(* IEC 61131-3 sources: crb-codesys/retrieval/output/codesys_repo/Proxy_Application/FUN, 9 files *)

(* ---- Proxy.st ---- *)
{attribute 'enable_dynamic_creation'}
FUNCTION_BLOCK Proxy IMPLEMENTS  Subject_Interface
VAR_INPUT
END_VAR
VAR_OUTPUT
END_VAR
VAR
	//Pointer to store the reference to the subject being protected
	refToRealSubject : POINTER TO Realsubject;
	//Last value of password entered by the client in the visualization element
	iTempPassword : INT;
END_VAR
VAR_STAT
	//Default password value for the request to be accepted
	iRealPassword : INT := 1234;
END_VAR

(* ---- Realsubject.st ---- *)
{attribute 'enable_dynamic_creation'}
FUNCTION_BLOCK Realsubject IMPLEMENTS  Subject_Interface
VAR_INPUT
END_VAR
VAR_OUTPUT
END_VAR
VAR
	//Variable to get and set values
	iProp: INT;
END_VAR

(* ---- Proxy_fb_init.st ---- *)
METHOD fb_init
VAR_INPUT
	//These boolean values are required for an automatic constructor
	bInitRetains : BOOL; // TRUE: the Retain-variables are initialized (reset warm / reset cold)
	bInCopyCode : BOOL;  // TRUE  the instance will be copied to the copy-code afterward (online change)

	//Pointer to the RealSubject instance
	ptrToRealSubject : POINTER TO Realsubject;
	//Local variable to store the password passed by the client with the password of the Proxy
	iTempPassword : INT;
	//Local variable to be used in WRITE request, it is the value to be set if the request is accepted
	iSetValue : INT;
	//Boolean value that specifies if the request is a WRITE or READ request
	bReadWrite : BOOL;
END_VAR
VAR_OUTPUT
END_VAR
VAR
	//Pointer to store the reference to the subject being protected
	refToRealSubject : POINTER TO Realsubject;
	//Last value of password entered by the client in the visualization element
	iTempPassword : INT;
END_VAR
VAR_STAT
	//Default password value for the request to be accepted
	iRealPassword : INT := 1234;
END_VAR

//Stores the address of the subject on a field in th Proxy.
THIS^.refToRealSubject := ptrToRealSubject;
//Stores the password value of the client on a field in the Proxy
THIS^.iTempPassword := iTempPassword;

//For security reasons, the Password passed by the client and the Proxi's connection password are compared
IF	THIS^.iTempPassword = THIS^.iRealPassword
	//If the password sent by the client is correct,
	THEN
	//We verify is the request is a SET or GET request
	IF bReadWrite
		//If the request is a SET request: boolean value TRUE
		THEN
		//The Proxy passes the request to the subject
		THIS^.Set_Method(iSetValue);
		//Once the request is completed, the Proxy responds to the client that the request has been accepted
		PLC_PRG.sTempSetLog := 'Request "SET" accepted';
		//If the request is a GET request: boolean value FALSE
		ELSE
		//The Proxy passes the request to the subject
		PLC_PRG.iGetValueLocal:= THIS^.Get_Method();
		//Once the request is completed, the Proxy responds to the client that the request has been accepted
		PLC_PRG.sTempGetLog := 'Request "GET" accepted';
	END_IF

	//If the password sent by the client is incorrect
	ELSE
	//We verify is the request is a SET or GET request
	IF bReadWrite
		//If the request is a SET request: boolean value TRUE
		THEN
		//The Proxy handles the bad request and response to the client without the subject intervention
		PLC_PRG.sTempSetLog := 'Request denied. Wrong password.';
		//If the request is a GET request: boolean value FALSE
		ELSE
		//The Proxy handles the bad request and response to the client without the subject intervention
		PLC_PRG.sTempGetLog := 'Request denied. Wrong password.';
	END_IF

END_IF

(* ---- Proxy_Get_Method.st ---- *)
METHOD Get_Method : INT
VAR_INPUT
END_VAR
VAR_OUTPUT
END_VAR
VAR
	//Pointer to store the reference to the subject being protected
	refToRealSubject : POINTER TO Realsubject;
	//Last value of password entered by the client in the visualization element
	iTempPassword : INT;
END_VAR
VAR_STAT
	//Default password value for the request to be accepted
	iRealPassword : INT := 1234;
END_VAR

Get_Method := THIS^.refToRealSubject^.Get_Method();

(* ---- Proxy_Set_Method.st ---- *)
METHOD Set_Method
VAR_INPUT
	//Value to be set to the subject passed as an input argument
	num	: INT;
END_VAR
VAR_OUTPUT
END_VAR
VAR
	//Pointer to store the reference to the subject being protected
	refToRealSubject : POINTER TO Realsubject;
	//Last value of password entered by the client in the visualization element
	iTempPassword : INT;
END_VAR
VAR_STAT
	//Default password value for the request to be accepted
	iRealPassword : INT := 1234;
END_VAR

THIS^.refToRealSubject^.Set_Method(num);

(* ---- Realsubject_Get_Method.st ---- *)
METHOD PUBLIC Get_Method : INT
VAR
	//Variable to get and set values
	iProp: INT;
END_VAR
Get_Method := THIS^.iProp;

(* ---- Realsubject_Set_Method.st ---- *)
METHOD Set_Method
VAR_INPUT
	//Value to be set on the iProp varible of realSubjectInstance
	num : INT;
    	//Variable to get and set values
	iProp: INT;
END_VAR

//Stores the value of the caller object on iProp variable.

THIS^.iProp := num;

(* ---- Subject_Interface_Get_Method.st ---- *)
METHOD Get_Method : int
VAR_INPUT
END_VAR

(* ---- Subject_Interface_Set_Method.st ---- *)
METHOD Set_Method
VAR_INPUT
	//Value to be set passed as an argument
	num : INT;
END_VAR
END_METHOD
